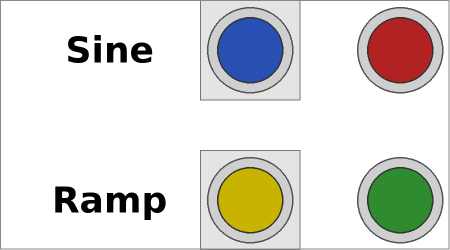
VISUALIZATION VISU_Program  // 450x250
    Lamp1 (350,150 100x100), variable: bLampRamp, style: Lamp-Lamp1-Green
    Lamp1 (350,0 100x100), variable: bLampSine, style: Lamp-Lamp1-Red
    PushSwitch (200,0 100x100), variable: bBtnSine, behaviour: TOGGLE, style: Switch-PushSwitch-Blue
    PushSwitch (200,150 100x100), variable: bBtnRamp, behaviour: TOGGLE, style: Switch-PushSwitch-Yellow
    Textfield (50,25 120x50), "Sine"
    Textfield (50,175 120x50), "Ramp"
END_VISUALIZATION

(* stored: Version 1.1.0.1
   Visu VISU_Program: Id {dcba0205-5e6c-48a7-a916-4849d8e906e3} *)
